(*
  Holds Marks definition & current state.
*)
{attribute 'no_explicit_call' := 'do not call this POU directly'} 
FUNCTION_BLOCK FB_MarkDefinition EXTENDS T_NamedBase IMPLEMENTS I_MarkDefinition
VAR
  // marks
  // - mark list
  _nMarks : UDINT;          // number of registered (teached) marks
  sMarkDef : ARRAY[1..200] OF ST_MarkDefinition;   // mark array (teached marks)
  
  // mark states
  _eMarkMode : E_MarkMode;
  _nMarksDetected : UDINT;  // number of detected marks

  // internals
  nMaxMarks : UDINT;
  sLastStartMark : ST_MarkDefinition;       // sampled start mark (because first mark will be overwritten already by next sheet)
  _a : LREAL;               // saved a Size
  
  // View
  _fImageLength, _fImageWidth, _fUseLength, _fDistBetweenMarks : LREAL;
  _nUses, _nMarksPerUse : UDINT;
  _bMarkInverted : BOOL;
  nSelMark : UDINT := 1;
  pSelMark : POINTER TO ST_MarkDefinition;
  bShowDetail : BOOL;
END_VAR
VAR CONSTANT
  // fixed triangle shape definition
  fC_MinUseLength     : LREAL := 0.04;  // minimal "use" length
  fC_MarkLengthMargin : LREAL := 0.1;   // [factor to a langth of mark] for mark length margin (to allow some jitter)
  //view
  nShSzX_px : UDINT := 700;
  nShSzY_px : UDINT := 180;
END_VAR

(*
  Definition of a mark.
  
   SqLength (1/2a or 2a) | TrLength = a -->
   |--------| \
   |        |   \
   |        |     \    -- center --
^  |        |       \
|  |--------|---------
| Height = a

Requirements:
  - StartMark has to be unique (bigger than minimal length of others)
  - Distance between Start and Endmark has to be bigger than length of StartMark + Minimal space
  - Mark has a minimum lenth, so the sensor can see the mark

*)

PROPERTY fMarkLengthMargin : LREAL
GET
fMarkLengthMargin := fC_MarkLengthMargin * _a;
END_GET
END_PROPERTY

(*
  Ge max length of marks.
*)
PROPERTY fMaxMarkLength : LREAL
GET
IF _nMarks > 0 THEN
  fMaxMarkLength := sMarkDef[1].fSqLength + sMarkDef[1].fTrLength;
END_IF
END_GET
END_PROPERTY

(*
  Get minimum length of hte start mark.
*)
PROPERTY fMinMarkLength : LREAL
GET
IF _nMarks > 0 THEN
  fMinMarkLength := sMarkDef[SEL(_nMarks>1, 1, 2)].fSqLength;
END_IF
END_GET
END_PROPERTY

(*
  Get a mark definition.
  nIdx= 1.._nMarks = registered marks
  nIdx= 0 - selects last mark 
  :returns: pointer to mark defintion or 0 if not found
*)
METHOD getMark : POINTER TO ST_MarkDefinition
VAR_INPUT
  nIdx : DINT; // mark index: 1.._nMarks, 0 = last (endMark) 
END_VAR
IF    nIdx = 0 THEN 
  getMark := ADR(sMarkDef[_nMarks]); // last mark (end or last)
ELSIF nIdx > 0 AND nIdx <= TO_DINT(_nMarks) THEN 
  getMark := ADR(sMarkDef[nIdx]);
ELSE 
  LogError(F_Concat2('Invalid mark requested, Idx=', TO_STRING(nIdx)));
END_IF
END_METHOD

METHOD Init : BOOL
VAR_INPUT
END_VAR
nMaxMarks := SIZEOF(sMarkDef) / SIZEOF(sMarkDef[1]);
ResetDefinition();
LogLevel := E_LogSeverity.Info;
END_METHOD

// return TRUE if its a StartMark
METHOD isStartMark : BOOL
VAR_INPUT
  fMarkLength : LREAL;    // mark length in [m]
END_VAR
IF _nMarks > 0 AND_THEN fMarkLength >= sMarkDef[1].fSqLength THEN  // square length of startMark
  isStartMark := TRUE;
END_IF
END_METHOD

(*Number of registered marks*)
PROPERTY nMarks : UDINT
GET
nMarks := _nMarks;
END_GET
END_PROPERTY

(*Number of detected marks*)
PROPERTY nMarksDetected : UDINT
GET
// number of detected marks
nMarksDetected := _nMarksDetected;
END_GET
END_PROPERTY

PROPERTY pLastStartMark : POINTER TO ST_MarkDefinition
GET
pLastStartMark := ADR(sLastStartMark);
END_GET
END_PROPERTY

(*
  Register a mark to camera (teach).
  If mark.nId >= 0 then it will be a detectable mark.
*)
METHOD RegisterMark : BOOL
VAR_INPUT
  sMark : ST_MarkDefinition;
END_VAR
VAR
  pMark : POINTER TO ST_MarkDefinition;
END_VAR
// - for all other teach marks
IF _nMarks >= nMaxMarks THEN LogError('Number of marks exeeded, ignore'); RETURN; END_IF
// we assume first mark is start mark, last mark is end mark (marks need to be registered in sorted order)
// (TODO) otherwise add marks in a sorted way to list
_nMarks := _nMarks + 1;
pMark := ADR(sMarkDef[_nMarks]);
// copy mark data
pMark^ := sMark;

// checks
// - set id if not given
IF pMark^.nId = 0 THEN pMark^.nId := TO_DINT(_nMarks); END_IF
// - start mark requirements
IF _nMarks > 1 THEN   
  // -- start mark length requirement 
  IF pMark^.fSqLength + pMark^.fTrLength >= sMarkDef[1].fSqLength THEN 
    LogError(F_Concat5('RegisterMark: mark not unique, too long: ', TO_STRING(pMark^.fSqLength + pMark^.fTrLength), ' > ', TO_STRING(sMarkDef[1].fSqLength), ' of start min. length'));
  END_IF
END_IF

// view
pMark^.sView.bShow := TRUE;
pMark^.sView.nXPosPx := TO_DINT(nShSzX_px*pMark^.fPosX/SEL(_fImageLength=0, _fImageLength, 1));
pMark^.sView.nYPosPx := TO_DINT(nShSzY_px*pMark^.fPosY/SEL(_fImageWidth=0,  _fImageWidth,  1));
pMark^.sView.colorFill := SEL(pMark^.nId=1, 16#FFAAABB6, 16#FF8E7CC3 );

// clear eventual mark state
MEMSET(destAddr:=ADR(pMark^.sState), 0, SIZEOF(ST_MarkState));

RegisterMark := TRUE;
END_METHOD

METHOD ResetDefinition
VAR
  i : UDINT;
END_VAR
ResetMarkStates();

_nMarks := 0;
_a := 0;

MEMSET(destAddr:=ADR(sMarkDef), fillByte:=0, SIZEOF(sMarkDef));
MEMSET(destAddr:=ADR(sLastStartMark), fillByte:=0, SIZEOF(sLastStartMark));
END_METHOD

(*
  Reset all registered marks
*)
METHOD ResetMarkStates
VAR
  i : UDINT;
END_VAR
// reset detected marks
_nMarksDetected := 0;
// reset mark state only
FOR i:=1 TO _nMarks DO
  MEMSET(destAddr:=ADR(sMarkDef[i].sState), 0, SIZEOF(ST_MarkState));
  sMarkDef[i].sView.colorFill := 16#FFFFFFFF;
END_FOR
//MEMSET(destAddr:=ADR(sLastStartMark.sState), 0, SIZEOF(ST_MarkState));
END_METHOD

METHOD saveMark : BOOL
VAR_INPUT
  pMark : POINTER TO ST_MarkDefinition;
END_VAR
IF pMark = 0 THEN RETURN; END_IF

IF NOT pMark^.sState.bMissed THEN
  pMark^.sView.colorFill := 16#FF7AF096; // (light greeen) 
ELSIF pMark^.sState.bMissed THEN 
  pMark^.sView.colorFill := 16#FFFD0000; // (some red)
END_IF

// sample start mark
IF pMark^.nId = 1 THEN 
  sLastStartMark := pMark^;           // save start mark as backup
  sMarkDef[pMark^.nId] := pMark^;     // save in teached mark table
  _nMarksDetected := _nMarksDetected + 1;
  saveMark := TRUE;

ELSIF pMark^.nId > 1 AND pMark^.nId <= TO_DINT(_nMarks) THEN
  sMarkDef[pMark^.nId] := pMark^;     // save in teached mark table
  _nMarksDetected := _nMarksDetected + 1;
  saveMark := TRUE;  
  
ELSE
  LogError(F_Concat3('saveMark: mark with id=', TO_STRING(pMark^.nId), ' not available'));
END_IF
END_METHOD

(*
  Calculate marks (position, shape) and register to mark definition. 
*)
METHOD PRIVATE TeachAuto : BOOL
VAR_INPUT
  a : LREAL;              // a length [m]
  c : LREAL;              // c start distance [m]
  bInverted : BOOL;       // mark inverted (flipped on x-axis)
END_VAR
VAR
  i : UDINT;
  bErr : BOOL;
  numMarks : UDINT;
  sNewMark : ST_MarkDefinition;
END_VAR

ResetDefinition();

// 
numMarks := _nUses*_nMarksPerUse;
IF numMarks = 0 THEN numMarks := 1; bErr:=TRUE; END_IF   // at least one mark
IF numMarks > 50 THEN numMarks:=50; bErr:=TRUE; LogError('TeachAuto: too many marks, limited to max. internal=50'); END_IF

_fDistBetweenMarks := _fImageLength/numMarks;

// calculate position
FOR i:=1 TO numMarks DO
  sNewMark.fHeight := a;
  sNewMark.fTrLength := a;
  sNewMark.fSqLength := SEL(i>1, 2*a, 0.5*a);
  sNewMark.fPosX := c + (i-1) * _fDistBetweenMarks;
  sNewMark.fPosY := 0;
  sNewMark.bInvertedX := bInverted;
  
  RegisterMark(sMark:=sNewMark);
END_FOR

TeachAuto := NOT bErr;
END_METHOD

(*Setup mark definition, teach marks for job x
  :return: TRUE if OK
*)
METHOD TeachMarks : BOOL
VAR_INPUT
  fImageLength             : LREAL := 1;      // Image length [m]
  fImageWidth              : LREAL := 1;      // Image width [m]
  eMarkMode                : E_MarkMode;      // mode for expected marks
  // mark format
  a       : LREAL;  // a= mark a length [m]
  b       : LREAL;  // b= mark a length [m]
  c       : LREAL;  // c= distance to start mark (from sheet border)
  nUses   : UDINT;  // use per repeat
  bMarkInverted  : BOOL;   // triangles are flipped Y
END_VAR
VAR
  bOk, bErr : BOOL;
END_VAR
_fImageLength := fImageLength;
_fImageWidth := fImageWidth;
_eMarkMode := eMarkMode;
_bMarkInverted := bMarkInverted;
_nUses := nUses;
_fUseLength := _fImageLength/nUses;
_nMarksPerUse := TO_UDINT(FLOOR(_fUseLength/fC_MinUseLength));
_a := a;

bOK := bErr := FALSE;

// checks
IF fImageLength/nUses < fC_MinUseLength THEN bErr:=TRUE; LogError('TeachMarks: Use length too small'); END_IF

// Teach new marks
IF    eMarkMode = E_MarkMode.AutoDefault THEN
  bOk := TeachAuto(a:=a, c:=c, bInverted:=bMarkInverted);
ELSIF eMarkMode = E_MarkMode.OneDefault THEN
  bOk := TeachOneMark(a:=a, c:=c, bInverted:=bMarkInverted);
ELSIF eMarkMode = E_MarkMode.OneTriangle THEN
  bOk := TeachOneTriangle(a:=a, b:=b, c:=c, bInverted:=bMarkInverted);
ELSIF eMarkMode = E_MarkMode.None THEN
  bOk := TeachOneSimMark();
END_IF

TeachMarks := bOk AND NOT bErr;
END_METHOD

(*
  Calculate marks (position, shape) and register to mark definition. 
*)
METHOD PRIVATE TeachOneMark : BOOL
VAR_INPUT
  a : LREAL;    // a length [m]
  c : LREAL;    // c start distance [m]
  bInverted : BOOL;
END_VAR
VAR
  sNewMark : ST_MarkDefinition;
END_VAR

ResetDefinition();

// > default mark (square & triangle)
// calculate position
sNewMark.fHeight := a;
sNewMark.fTrLength := a;
sNewMark.fSqLength := 2 * a;
sNewMark.fPosX := c;
sNewMark.fPosY := 0;
sNewMark.bInvertedX := bInverted;

RegisterMark(sMark:=sNewMark);

TeachOneMark := TRUE;
END_METHOD

(*
  Calculate marks (position, shape) and register to mark definition. 
*)
METHOD PRIVATE TeachOneSimMark : BOOL
VAR_INPUT
END_VAR
VAR
  sNewMark : ST_MarkDefinition;
END_VAR

ResetDefinition();

// > a simulation/generation mark
// calculate position
sNewMark.bVirtual := TRUE;
sNewMark.fHeight := 0.001;
sNewMark.fTrLength := 0.001;
sNewMark.fSqLength := 0;
sNewMark.fPosX := 0;
sNewMark.fPosY := 0;
sNewMark.bInvertedX := FALSE;

RegisterMark(sMark:=sNewMark);

TeachOneSimMark := TRUE;
END_METHOD

(*
  Calculate marks (position, shape) and register to mark definition. 
*)
METHOD PRIVATE TeachOneTriangle : BOOL
VAR_INPUT
  a : LREAL;    // a length [m]
  b : LREAL;    // b length [m]
  c : LREAL;    // c start distance [m]
  bInverted : BOOL;
END_VAR
VAR
  sNewMark : ST_MarkDefinition;
END_VAR

ResetDefinition();

// calculate position
// > triangle only  (squareLen=0)
sNewMark.fHeight := a;
sNewMark.fTrLength := b;
sNewMark.fSqLength := 0;
sNewMark.fPosX := c;
sNewMark.fPosY := 0;
sNewMark.bInvertedX := bInverted;  

RegisterMark(sMark:=sNewMark);

TeachOneTriangle := TRUE;
END_METHOD

METHOD update_view
VAR_INPUT
END_VAR
nSelMark := LIMIT(1, nSelMark, nMaxMarks);
pSelMark := ADR(sMarkDef[nSelMark]);
END_METHOD

END_FUNCTION_BLOCK

(* stored: Version 1.1.0.1, ProductVersion 3.1.4024.11
   POU FB_MarkDefinition: Id {9fd490d8-a121-44dc-9636-b7387d840542}, SpecialFunc None
   Folder I_MarkDefinition: Id {768d0757-a8ce-42f3-be27-86b1dccd832c}
   Folder Teaching: Id {d7f1a474-7ab0-4d97-9fc3-29f084e73191}
   Property fMarkLengthMargin: Id {6354683d-c554-4595-afc5-0b4ee6712206}
   Get Get: Id {aee51c4d-dbff-4339-bb35-85ed5d0cc192}
   Property fMaxMarkLength: Id {43ac1333-9baa-4872-95db-9700173f90dd}
   Get Get: Id {a57cf7c0-a0b4-4e15-a8a7-8af41d7a28e0}
   Property fMinMarkLength: Id {28ad9750-49f7-4210-8ae8-7698496aabf2}
   Get Get: Id {fde96c83-e5b8-4ed6-ab57-405d7b3125a8}
   Method getMark: Id {c37a739d-c91b-4a27-ba64-795297055335}
   Method Init: Id {10e5662f-25fc-4596-8060-c14e2fb3ea29}
   Method isStartMark: Id {3e3e599f-4d3b-4e89-be04-2c96b56f1dec}
   Property nMarks: Id {d1a014db-64d0-4106-adc4-b24435d88146}
   Get Get: Id {754530ed-d7a4-4c92-bf61-956c368cbf56}
   Property nMarksDetected: Id {d8225d80-c29e-447c-bdae-b0ba98c5da47}
   Get Get: Id {88f4a7a9-ca4b-4f17-b72f-9481bb832a9a}
   Property pLastStartMark: Id {9dfa6397-d969-4853-8cda-cff0a6683302}
   Get Get: Id {d6dce974-ba32-4a91-8230-fe6e741ba47b}
   Method RegisterMark: Id {8567991f-e325-4655-876e-2d25aa46922c}
   Method ResetDefinition: Id {aca53e14-0a95-43b2-9963-e58fc6977ee5}
   Method ResetMarkStates: Id {028fa150-b018-4ff3-b9f7-6a74efb6afb2}
   Method saveMark: Id {b829c69e-69eb-412a-a77a-9b1cda33bddd}
   Method TeachAuto: Id {d881e1d3-0f3e-4142-90f4-761a524a5ce0}
   Method TeachMarks: Id {0862f9ff-112d-4178-95a2-88b41209d52d}
   Method TeachOneMark: Id {b29aa47a-aa65-45ec-a32e-d33a1e8344f2}
   Method TeachOneSimMark: Id {453a94e7-603c-485c-9e23-e7ac2a920742}
   Method TeachOneTriangle: Id {c2c1a8d2-eed4-4e97-9356-e7bcd531caed}
   Method update_view: Id {41a8142f-4950-483a-a733-e026dfe68780} *)
